// Mitsubishi GX Developer project: Закатка(LOLLETTE)   PLC: FX3U

PROGRAM MAIN
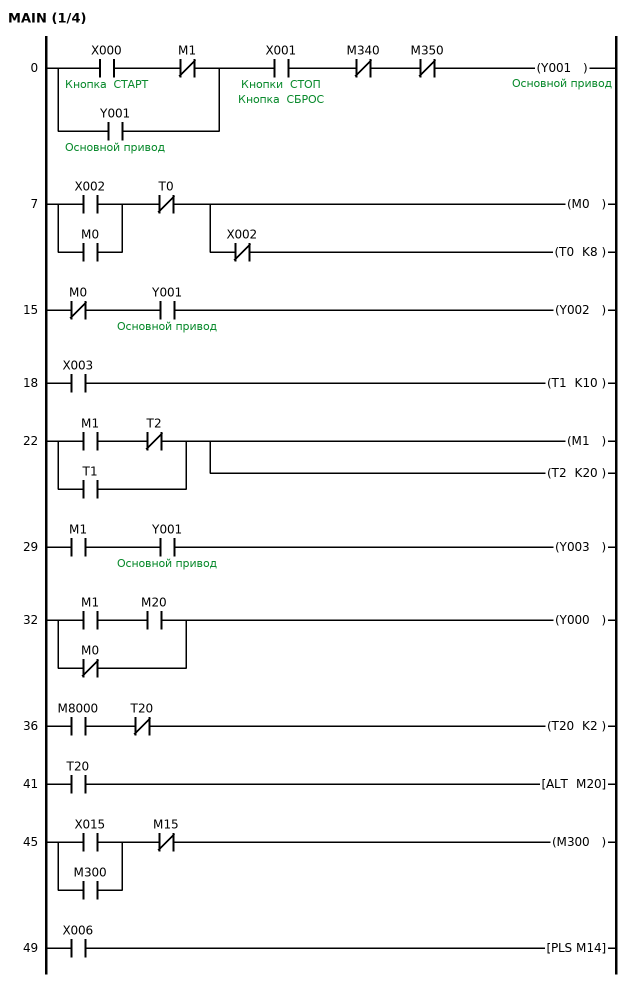
0     LD      X000  ; Кнопка  СТАРТ
      ANI     M1
      OR      Y001  ; Основной привод
      AND     X001  ; Кнопки  СТОП    Кнопка  СБРОС
      ANI     M340
      ANI     M350
      OUT     Y001  ; Основной привод
7     LD      X002
      OR      M0
      ANI     T0
      OUT     M0
      ANI     X002
      OUT     T0 K8
15    LDI     M0
      AND     Y001  ; Основной привод
      OUT     Y002
18    LD      X003
      OUT     T1 K10
22    LD      M1
      ANI     T2
      OR      T1
      OUT     M1
      OUT     T2 K20
29    LD      M1
      AND     Y001  ; Основной привод
      OUT     Y003
32    LD      M1
      AND     M20
      ORI     M0
      OUT     Y000
36    LD      M8000
      ANI     T20
      OUT     T20 K2
41    LD      T20
      ALT     M20
45    LD      X015
      OR      M300
      ANI     M15
      OUT     M300
49    LD      X006
      PLS     M14
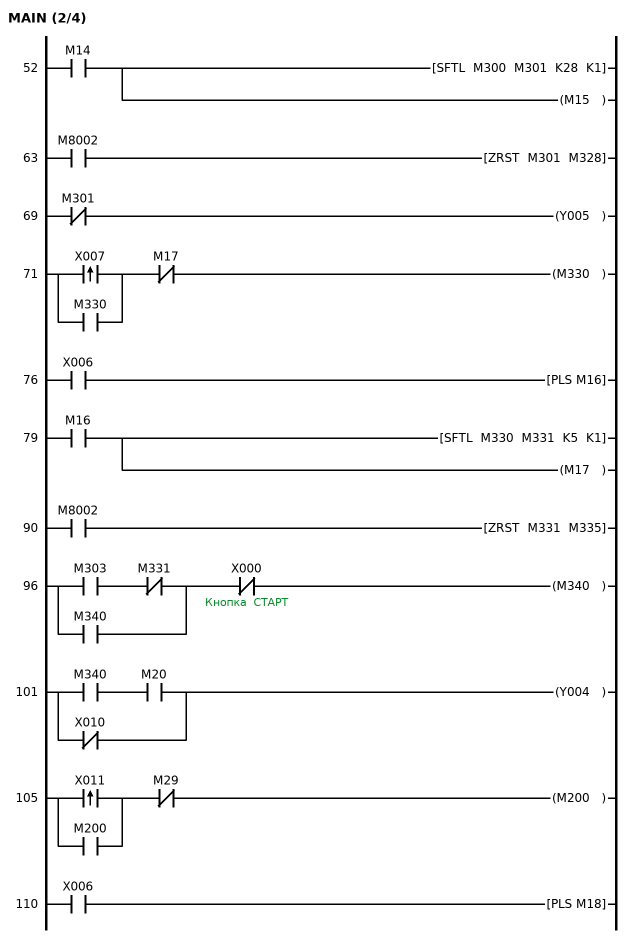
52    LD      M14
      SFTL    M300 M301 K28 K1
      OUT     M15
63    LD      M8002
      ZRST    M301 M328
69    LDI     M301
      OUT     Y005
71    LDP     X007
      OR      M330
      ANI     M17
      OUT     M330
76    LD      X006
      PLS     M16
79    LD      M16
      SFTL    M330 M331 K5 K1
      OUT     M17
90    LD      M8002
      ZRST    M331 M335
96    LD      M303
      ANI     M331
      OR      M340
      ANI     X000  ; Кнопка  СТАРТ
      OUT     M340
101   LD      M340
      AND     M20
      ORI     X010
      OUT     Y004
105   LDP     X011
      OR      M200
      ANI     M29
      OUT     M200
110   LD      X006
      PLS     M18
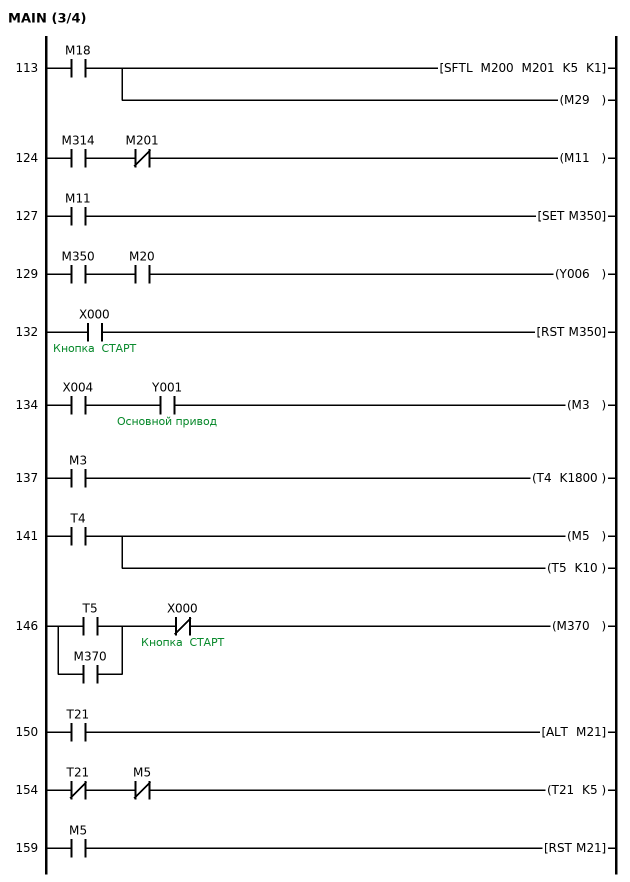
113   LD      M18
      SFTL    M200 M201 K5 K1
      OUT     M29
124   LD      M314
      ANI     M201
      OUT     M11
127   LD      M11
      SET     M350
129   LD      M350
      AND     M20
      OUT     Y006
132   LD      X000  ; Кнопка  СТАРТ
      RST     M350
134   LD      X004
      AND     Y001  ; Основной привод
      OUT     M3
137   LD      M3
      OUT     T4 K1800
141   LD      T4
      OUT     M5
      OUT     T5 K10
146   LD      T5
      OR      M370
      ANI     X000  ; Кнопка  СТАРТ
      OUT     M370
150   LD      T21
      ALT     M21
154   LDI     T21
      ANI     M5
      OUT     T21 K5
159   LD      M5
      RST     M21
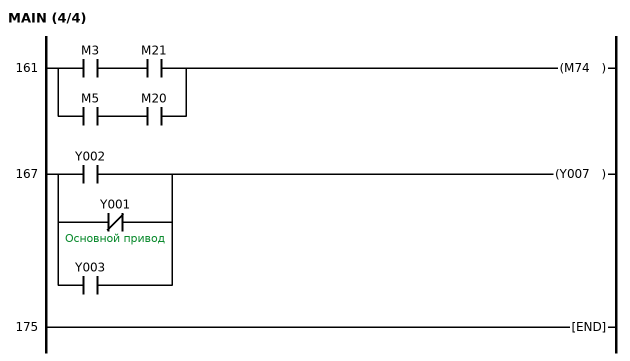
161   LD      M3
      AND     M21
      LD      M5
      AND     M20
      ORB
      OUT     M74
167   LD      Y002
      ORI     Y001  ; Основной привод
      OR      Y003
      OUT     Y007
175   END
END_PROGRAM
